PROGRAM MAIN
VAR
	trafficLight_1			: FB_TrafficLight;
	
	// control variables
	clear					: BOOL;
	block					: BOOL;
	disable					: BOOL;
	
	// output variables
	red						: BOOL;
	yellow					: BOOL;
	green					: BOOL;
END_VAR

trafficLight_1(clear_road := clear, block_road := block, disable_system := disable);

red := trafficLight_1.red_light;
yellow := trafficLight_1.yellow_light;
green := trafficLight_1.green_light;

END_PROGRAM

(* stored: Version 1.1.0.1, ProductVersion 3.1.4024.9
   POU MAIN: Id {1a1fe5cd-92b2-4c7c-b7fc-d151960b93c6}, SpecialFunc None *)
